// TIA Portal project "FESTO_SORTING_AND_DISTRIBUTING_STATION_WITH_HMI_AND_SCALANCE_V17_1" (V17)

(* hardware
DEVICE "S71500/ET200MP station_1"  S7-1500 station
   slot 0: "Rail_0"  Rack  6ES7 590-1***0-0AA0
   slot 1: "Sorting Station"  CPU 1512C-1 PN  6ES7 512-1CK01-0AB0  V2.5
      slot 3: "CPU display_1"  6ES7591-1AA00-0AA0
      slot 32768: "PROFINET interface_1"  X1
         slot 32769: "Port_1"  X1 P1
         slot 32770: "Port_2"  X1 P2
DEVICE "S71500/ET200MP station_2"  S7-1500 station
   slot 0: "Rail_0"  Rack  6ES7 590-1***0-0AA0
   slot 1: "Distributing Station"  CPU 1512C-1 PN  6ES7 512-1CK01-0AB0  V2.5
      slot 3: "CPU display_1"  6ES7591-1AA00-0AA0
      slot 32768: "PROFINET interface_1"  X1
         slot 32769: "Port_1"  X1 P1
         slot 32770: "Port_2"  X1 P2
DEVICE "HMI_1"  TP700 Comfort
   slot 0: "HMI_1"  TP700 Comfort  6AV2 124-0GC01-0AX0  16.0.0.0
   slot 1: "HMI_RT_1"  TP700 Comfort  6AV2 124-0GC01-0AX0  16.0.0.0
   slot 5: "HMI_1.IE_CP_1"  PROFINET Interface  16.0.0.0
      slot 1: "PROFINET Interface_1"  PROFINET Interface
         slot 1: "Port_1"  Port
         slot 2: "Port_2"  Port
   slot 7: "HMI_1.MPI/DP_CP_1"  MPI/DP Interface  16.0.0.0
*)

// ===== PLC "Sorting Station"  CPU 1512C-1 PN =====

VAR_GLOBAL   // PLC tag table "Default tag table"
   "ITEM_COUNTER_(PHOTOELECTRIC)" AT %I1.0 : Bool;
   "SORTER_EXTENDED_(INDUCTIVE)" AT %I1.1 : Bool;
   "CONVEYER" AT %Q5.2 : Bool;
   "SORTER" AT %Q5.0 : Bool;
   "START" AT %I0.0 : Bool;
   "STOP" AT %I0.1 : Bool;
   "AUTO" AT %I0.2 : Bool;
   "RESET" AT %I0.3 : Bool;
   "HMI_START" AT %M20.0 : Bool;
   "HMI_STOP" AT %M20.1 : Bool;
   "HMI_RESET" AT %M20.2 : Bool;
   "HMI_AUTO" AT %M20.3 : Bool;
   "POWER" AT %M0.0 : Bool;
   "BLACK_PART_MEM" AT %M40.0 : Bool;
   "PINK_PART_MEM" AT %M40.1 : Bool;
   "Clock_Byte" AT %MB300 : Byte;
   "Clock_10Hz" AT %M300.0 : Bool;
   "Clock_5Hz" AT %M300.1 : Bool;
   "Clock_2.5Hz" AT %M300.2 : Bool;
   "Clock_2Hz" AT %M300.3 : Bool;
   "Clock_1.25Hz" AT %M300.4 : Bool;
   "Clock_1Hz" AT %M300.5 : Bool;
   "Clock_0.625Hz" AT %M300.6 : Bool;
   "Clock_0.5Hz" AT %M300.7 : Bool;
   "Tag_1" AT %M40.2 : Bool;
   "RESTART_MEM" AT %M40.4 : Bool;
END_VAR

DATA_BLOCK "STEPS"   // DB2
{ S7_Optimized_Access := 'TRUE' }
VERSION : 0.1
   VAR
      Current_Step : Int;
   END_VAR
BEGIN
END_DATA_BLOCK

// folder: System blocks/Program resources

DATA_BLOCK "IEC_Timer_0_DB"   // DB3
{ S7_Optimized_Access := 'TRUE' }
AUTHOR : Simatic
FAMILY : IEC
NAME : IEC_TMR
VERSION : 1.0
// stored: InstanceOfName IEC_TIMER
"IEC_TIMER"
BEGIN
END_DATA_BLOCK

// folder: (top level)

ORGANIZATION_BLOCK "Sorting"   // OB1, LAD, ProgramCycle
TITLE = "Main Program Sweep (Cycle)"
{ S7_Optimized_Access := 'TRUE' }
VERSION : 0.1
   VAR_INPUT
      Initial_Call : Bool;   // Initial call of this OB
      Remanence : Bool;   // =True, if remanent data are available
   END_VAR
   VAR_TEMP   // added for the SCL form of the ladder/FBD networks
      _w1 : Bool;
      _w2 : Bool;
      _w3 : Bool;
   END_VAR
BEGIN

REGION Network 1
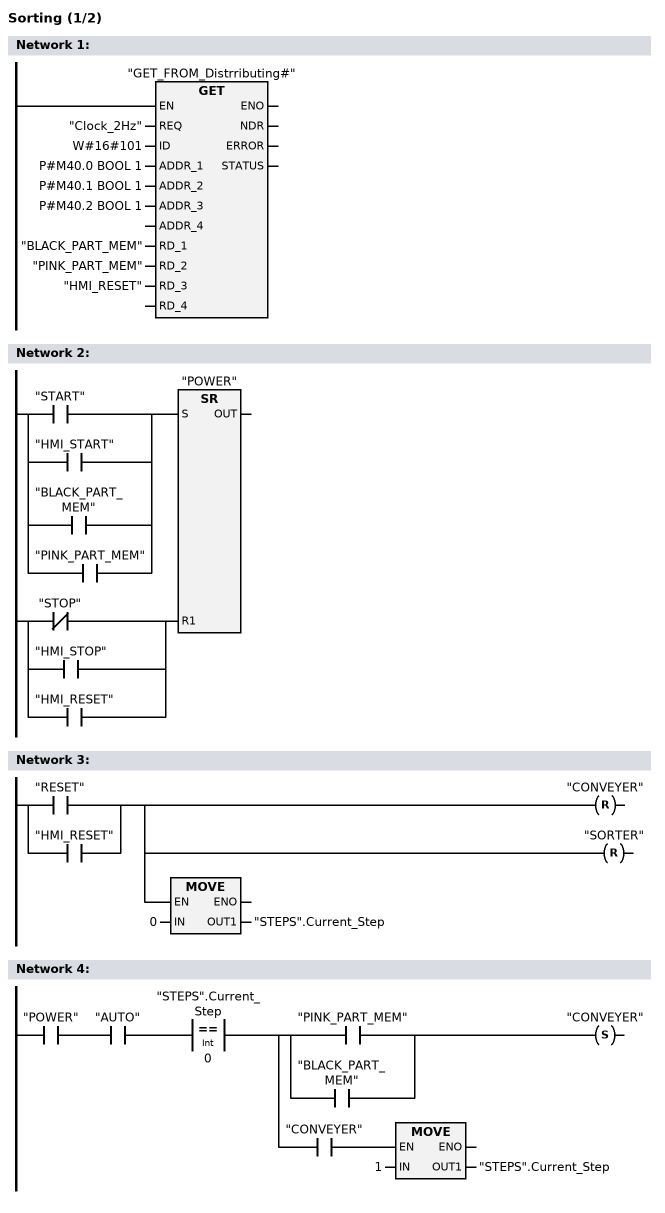
   "GET_FROM_Distrributing#"(REQ := "Clock_2Hz",   // GET
                           ID := W#16#101,
                           ADDR_1 := P#M40.0 BOOL 1,
                           ADDR_2 := P#M40.1 BOOL 1,
                           ADDR_3 := P#M40.2 BOOL 1,
                           RD_1 := "BLACK_PART_MEM",
                           RD_2 := "PINK_PART_MEM",
                           RD_3 := "HMI_RESET");
END_REGION

REGION Network 2
   RUNG wire#powerrail
      Contact( "START" )
      wire#w1
      S_SR(operand := "POWER", r1 := wire#w2)
   END_RUNG
   RUNG wire#powerrail
      Contact( "HMI_START" )
   END_RUNG wire#w1
   RUNG wire#powerrail
      Contact( "BLACK_PART_MEM" )
   END_RUNG wire#w1
   RUNG wire#powerrail
      Contact( "PINK_PART_MEM" )
   END_RUNG wire#w1
   RUNG wire#powerrail
      I_Contact( "STOP" )
   END_RUNG wire#w2
   RUNG wire#powerrail
      Contact( "HMI_STOP" )
   END_RUNG wire#w2
   RUNG wire#powerrail
      Contact( "HMI_RESET" )
   END_RUNG wire#w2
   // the same network as SCL:
   IF "START" OR "HMI_START" OR "BLACK_PART_MEM" OR "PINK_PART_MEM" THEN
       "POWER" := TRUE;   // SR flip-flop
   END_IF;
   IF NOT "STOP" OR "HMI_STOP" OR "HMI_RESET" THEN "POWER" := FALSE; END_IF;
END_REGION

REGION Network 3
   RUNG wire#powerrail
      Contact( "RESET" )
      wire#w1
      R_Coil( "CONVEYER" )
   END_RUNG
   RUNG wire#powerrail
      Contact( "HMI_RESET" )
   END_RUNG wire#w1
   RUNG wire#w1
      R_Coil( "SORTER" )
   END_RUNG
   RUNG wire#w1
      Move(in := 0, out1 => "STEPS".Current_Step)
   END_RUNG
   // the same network as SCL:
   IF "RESET" OR "HMI_RESET" THEN
       "CONVEYER" := FALSE;
       "SORTER" := FALSE;
       "STEPS".Current_Step := 0;
   END_IF;
END_REGION

REGION Network 4
   RUNG wire#powerrail
      Contact( "POWER" )
      Contact( "AUTO" )
      { S7_Templates := "SrcType := Int" } EQ_Contact(in1 := "STEPS".Current_Step, in2 := 0)
      wire#w1
      Contact( "PINK_PART_MEM" )
      wire#w2
      S_Coil( "CONVEYER" )
   END_RUNG
   RUNG wire#w1
      Contact( "BLACK_PART_MEM" )
   END_RUNG wire#w2
   RUNG wire#w1
      Contact( "CONVEYER" )
      Move(in := 1, out1 => "STEPS".Current_Step)
   END_RUNG
   // the same network as SCL:
   #_w1 := "POWER" AND "AUTO" AND ("STEPS".Current_Step = 0);
   IF #_w1 AND ("PINK_PART_MEM" OR "BLACK_PART_MEM") THEN "CONVEYER" := TRUE; END_IF;
   IF #_w1 AND "CONVEYER" THEN "STEPS".Current_Step := 1; END_IF;
END_REGION

REGION Network 5
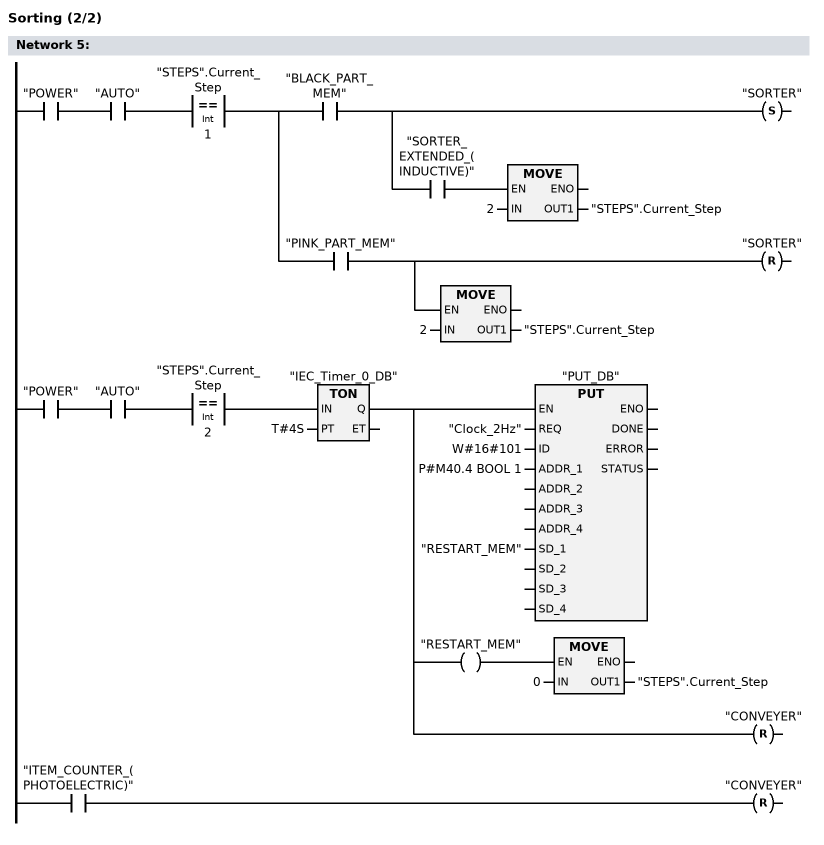
   #_w1 := "POWER" AND "AUTO" AND ("STEPS".Current_Step = 1);
   #_w2 := #_w1 AND "BLACK_PART_MEM";
   IF #_w2 THEN "SORTER" := TRUE; END_IF;
   IF #_w2 AND "SORTER_EXTENDED_(INDUCTIVE)" THEN "STEPS".Current_Step := 2; END_IF;
   IF #_w1 AND "PINK_PART_MEM" THEN
       "SORTER" := FALSE;
       "STEPS".Current_Step := 2;
   END_IF;
   "IEC_Timer_0_DB".TON(IN := "POWER" AND "AUTO" AND ("STEPS".Current_Step = 2), PT := T#4S);
   #_w3 := "IEC_Timer_0_DB".Q;
   IF #_w3 THEN
       "PUT_DB"(REQ := "Clock_2Hz", ID := W#16#101, ADDR_1 := P#M40.4 BOOL 1, SD_1 := "RESTART_MEM");   // PUT
   END_IF;
   "RESTART_MEM" := #_w3;
   IF #_w3 THEN
       "STEPS".Current_Step := 0;
       "CONVEYER" := FALSE;
   END_IF;
   IF "ITEM_COUNTER_(PHOTOELECTRIC)" THEN "CONVEYER" := FALSE; END_IF;
END_REGION
END_ORGANIZATION_BLOCK

// ===== PLC "Distributing Station"  CPU 1512C-1 PN =====

VAR_GLOBAL   // PLC tag table "Default tag table"
   "START" AT %I0.0 : Bool;
   "STOP" AT %I0.1 : Bool;
   "AUTO" AT %I0.2 : Bool;
   "RESET" AT %I0.3 : Bool;
   "PART_PRESENT(SORTING)" AT %I1.4 : Bool;
   "PHOTOELECTRIC(differentiate btwn black and pink)" AT %I1.7 : Bool;
   "INDUCTIVE(metallic and non-metallic" AT %I1.6 : Bool;
   "FEED_CYLINDER_EXTENDED" AT %I1.0 : Bool;
   "SORTER_EXTENDED" AT %I1.3 : Bool;
   "PART_PRESENT(FEED_CYLINDER)" AT %I1.2 : Bool;
   "HMI_START" AT %M0.0 : Bool;
   "HMI_STOP" AT %M0.1 : Bool;
   "HMI_AUTO" AT %M0.2 : Bool;
   "HMI_RESET" AT %M0.3 : Bool;
   "POWER" AT %M100.0 : Bool;
   "AUTO_MEM" AT %M100.1 : Bool;
   "CONVEYER_BACKWARD" AT %Q5.3 : Bool;
   "EXTEND_FEED_CYLINDER" AT %Q5.1 : Bool;
   "SORTER" AT %Q5.2 : Bool;
   "CONVEYER_FORWARD" AT %Q5.0 : Bool;
   "PART_HOLDER" AT %Q5.5 : Bool;
   "BLACK_MEM" AT %M40.0 : Bool;
   "PINK_MEM" AT %M40.1 : Bool;
   "Clock_Byte" AT %MB300 : Byte;
   "Clock_10Hz" AT %M300.0 : Bool;
   "Clock_5Hz" AT %M300.1 : Bool;
   "Clock_2.5Hz" AT %M300.2 : Bool;
   "Clock_2Hz" AT %M300.3 : Bool;
   "Clock_1.25Hz" AT %M300.4 : Bool;
   "Clock_1Hz" AT %M300.5 : Bool;
   "Clock_0.625Hz" AT %M300.6 : Bool;
   "Clock_0.5Hz" AT %M300.7 : Bool;
   "HMI_LED_RESET" AT %M100.4 : Bool;
   "STOP_MEM" AT %M100.5 : Bool;
   "RESET_MEM" AT %M40.2 : Bool;
   "Tag_1" AT %M20.2 : Bool;
   "RESTART_MEM" AT %M40.4 : Bool;
END_VAR

DATA_BLOCK "STEPS"   // DB1
{ S7_Optimized_Access := 'TRUE' }
VERSION : 0.1
   VAR
      Current_Steps : Real;
   END_VAR
BEGIN
END_DATA_BLOCK

// folder: System blocks/Program resources

DATA_BLOCK "#"   // DB2
{ S7_Optimized_Access := 'TRUE' }
AUTHOR : Simatic
FAMILY : IEC
NAME : IEC_TMR
VERSION : 1.0
// stored: InstanceOfName IEC_TIMER
"IEC_TIMER"
BEGIN
END_DATA_BLOCK

DATA_BLOCK "IEC_Timer_0_DB"   // DB5
{ S7_Optimized_Access := 'TRUE' }
AUTHOR : Simatic
FAMILY : IEC
NAME : IEC_TMR
VERSION : 1.0
// stored: InstanceOfName IEC_TIMER
"IEC_TIMER"
BEGIN
END_DATA_BLOCK

DATA_BLOCK "IEC_Timer_0_DB_1"   // DB8
{ S7_Optimized_Access := 'TRUE' }
AUTHOR : Simatic
FAMILY : IEC
NAME : IEC_TMR
VERSION : 1.0
// stored: InstanceOfName IEC_TIMER
"IEC_TIMER"
BEGIN
END_DATA_BLOCK

DATA_BLOCK "IEC_Timer_0_DB_2"   // DB9
{ S7_Optimized_Access := 'TRUE' }
AUTHOR : Simatic
FAMILY : IEC
NAME : IEC_TMR
VERSION : 1.0
// stored: InstanceOfName IEC_TIMER
"IEC_TIMER"
BEGIN
END_DATA_BLOCK

// folder: (top level)

ORGANIZATION_BLOCK "Distributing"   // OB1, LAD, ProgramCycle
TITLE = "Main Program Sweep (Cycle)"
{ S7_Optimized_Access := 'TRUE' }
VERSION : 0.1
   VAR_INPUT
      Initial_Call : Bool;   // Initial call of this OB
      Remanence : Bool;   // =True, if remanent data are available
   END_VAR
   VAR_TEMP   // added for the SCL form of the ladder/FBD networks
      _w1 : Bool;
      _w2 : Bool;
   END_VAR
BEGIN

REGION Network 1
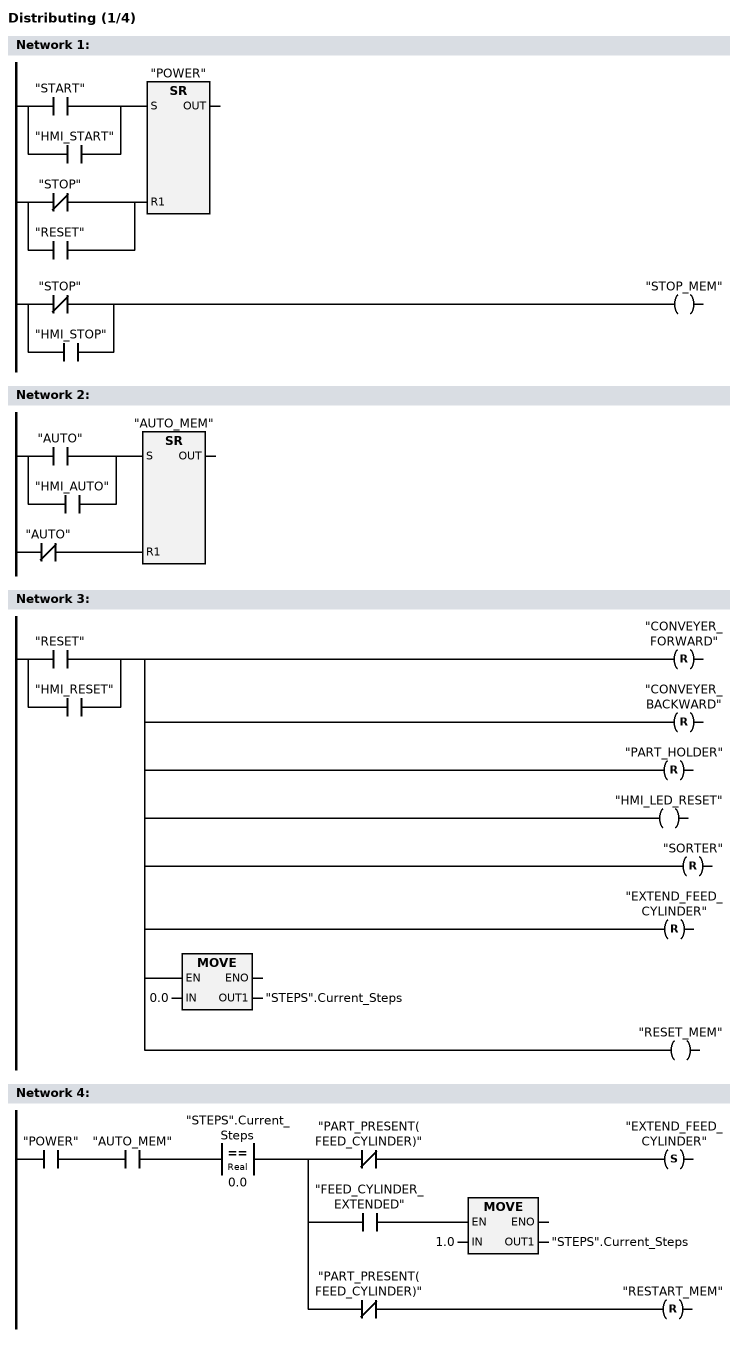
   RUNG wire#powerrail
      Contact( "START" )
      wire#w1
      S_SR(operand := "POWER", r1 := wire#w2)
   END_RUNG
   RUNG wire#powerrail
      Contact( "HMI_START" )
   END_RUNG wire#w1
   RUNG wire#powerrail
      I_Contact( "STOP" )
   END_RUNG wire#w2
   RUNG wire#powerrail
      Contact( "RESET" )
   END_RUNG wire#w2
   RUNG wire#powerrail
      I_Contact( "STOP" )
      wire#w3
      Coil( "STOP_MEM" )
   END_RUNG
   RUNG wire#powerrail
      Contact( "HMI_STOP" )
   END_RUNG wire#w3
   // the same network as SCL:
   IF "START" OR "HMI_START" THEN
       "POWER" := TRUE;   // SR flip-flop
   END_IF;
   IF NOT "STOP" OR "RESET" THEN "POWER" := FALSE; END_IF;
   "STOP_MEM" := NOT "STOP" OR "HMI_STOP";
END_REGION

REGION Network 2
   RUNG wire#powerrail
      Contact( "AUTO" )
      wire#w1
      S_SR(operand := "AUTO_MEM", r1 := wire#w2)
   END_RUNG
   RUNG wire#powerrail
      Contact( "HMI_AUTO" )
   END_RUNG wire#w1
   RUNG wire#powerrail
      I_Contact( "AUTO" )
   END_RUNG wire#w2
   // the same network as SCL:
   IF "AUTO" OR "HMI_AUTO" THEN
       "AUTO_MEM" := TRUE;   // SR flip-flop
   END_IF;
   IF NOT "AUTO" THEN "AUTO_MEM" := FALSE; END_IF;
END_REGION

REGION Network 3
   RUNG wire#powerrail
      Contact( "RESET" )
      wire#w1
      R_Coil( "CONVEYER_FORWARD" )
   END_RUNG
   RUNG wire#powerrail
      Contact( "HMI_RESET" )
   END_RUNG wire#w1
   RUNG wire#w1
      R_Coil( "CONVEYER_BACKWARD" )
   END_RUNG
   RUNG wire#w1
      R_Coil( "PART_HOLDER" )
   END_RUNG
   RUNG wire#w1
      Coil( "HMI_LED_RESET" )
   END_RUNG
   RUNG wire#w1
      R_Coil( "SORTER" )
   END_RUNG
   RUNG wire#w1
      R_Coil( "EXTEND_FEED_CYLINDER" )
   END_RUNG
   RUNG wire#w1
      Move(in := 0.0, out1 => "STEPS".Current_Steps)
   END_RUNG
   RUNG wire#w1
      Coil( "RESET_MEM" )
   END_RUNG
   // the same network as SCL:
   #_w1 := "RESET" OR "HMI_RESET";
   IF #_w1 THEN
       "CONVEYER_FORWARD" := FALSE;
       "CONVEYER_BACKWARD" := FALSE;
       "PART_HOLDER" := FALSE;
   END_IF;
   "HMI_LED_RESET" := #_w1;
   IF #_w1 THEN
       "SORTER" := FALSE;
       "EXTEND_FEED_CYLINDER" := FALSE;
       "STEPS".Current_Steps := 0.0;
   END_IF;
   "RESET_MEM" := #_w1;
END_REGION

REGION Network 4
   RUNG wire#powerrail
      Contact( "POWER" )
      Contact( "AUTO_MEM" )
      { S7_Templates := "SrcType := Real" } EQ_Contact(in1 := "STEPS".Current_Steps, in2 := 0.0)
      wire#w1
      I_Contact( "PART_PRESENT(FEED_CYLINDER)" )
      S_Coil( "EXTEND_FEED_CYLINDER" )
   END_RUNG
   RUNG wire#w1
      Contact( "FEED_CYLINDER_EXTENDED" )
      Move(in := 1.0, out1 => "STEPS".Current_Steps)
   END_RUNG
   RUNG wire#w1
      I_Contact( "PART_PRESENT(FEED_CYLINDER)" )
      R_Coil( "RESTART_MEM" )
   END_RUNG
   // the same network as SCL:
   #_w1 := "POWER" AND "AUTO_MEM" AND ("STEPS".Current_Steps = 0.0);
   IF #_w1 AND NOT "PART_PRESENT(FEED_CYLINDER)" THEN "EXTEND_FEED_CYLINDER" := TRUE; END_IF;
   IF #_w1 AND "FEED_CYLINDER_EXTENDED" THEN "STEPS".Current_Steps := 1.0; END_IF;
   IF #_w1 AND NOT "PART_PRESENT(FEED_CYLINDER)" THEN "RESTART_MEM" := FALSE; END_IF;
END_REGION

REGION Network 5
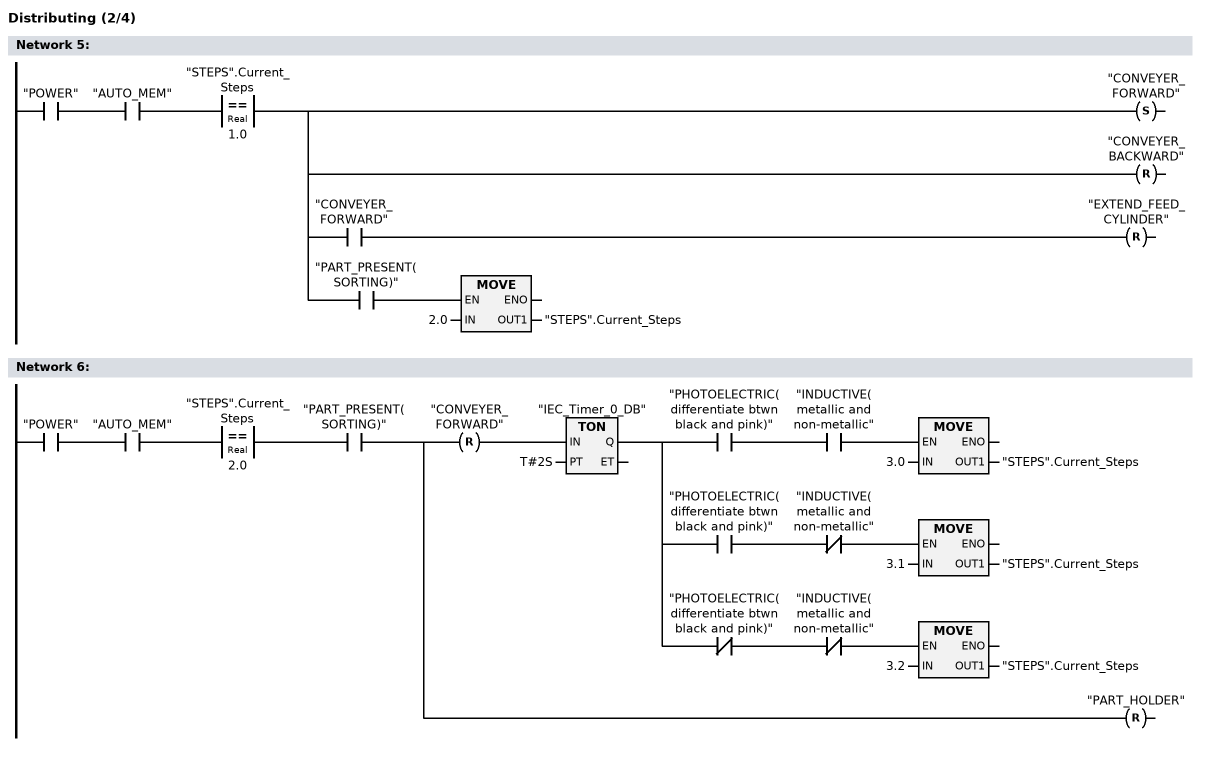
   RUNG wire#powerrail
      Contact( "POWER" )
      Contact( "AUTO_MEM" )
      { S7_Templates := "SrcType := Real" } EQ_Contact(in1 := "STEPS".Current_Steps, in2 := 1.0)
      wire#w1
      S_Coil( "CONVEYER_FORWARD" )
   END_RUNG
   RUNG wire#w1
      R_Coil( "CONVEYER_BACKWARD" )
   END_RUNG
   RUNG wire#w1
      Contact( "CONVEYER_FORWARD" )
      R_Coil( "EXTEND_FEED_CYLINDER" )
   END_RUNG
   RUNG wire#w1
      Contact( "PART_PRESENT(SORTING)" )
      Move(in := 2.0, out1 => "STEPS".Current_Steps)
   END_RUNG
   // the same network as SCL:
   #_w1 := "POWER" AND "AUTO_MEM" AND ("STEPS".Current_Steps = 1.0);
   IF #_w1 THEN
       "CONVEYER_FORWARD" := TRUE;
       "CONVEYER_BACKWARD" := FALSE;
   END_IF;
   IF #_w1 AND "CONVEYER_FORWARD" THEN "EXTEND_FEED_CYLINDER" := FALSE; END_IF;
   IF #_w1 AND "PART_PRESENT(SORTING)" THEN "STEPS".Current_Steps := 2.0; END_IF;
END_REGION

REGION Network 6
   #_w1 := "POWER" AND "AUTO_MEM" AND ("STEPS".Current_Steps = 2.0) AND "PART_PRESENT(SORTING)";
   IF #_w1 THEN "CONVEYER_FORWARD" := FALSE; END_IF;
   "IEC_Timer_0_DB".TON(IN := #_w1, PT := T#2S);
   IF "IEC_Timer_0_DB".Q AND "PHOTOELECTRIC(differentiate btwn black and pink)" AND "INDUCTIVE(metallic and non-metallic" THEN
       "STEPS".Current_Steps := 3.0;
   END_IF;
   IF "IEC_Timer_0_DB".Q AND "PHOTOELECTRIC(differentiate btwn black and pink)" AND NOT "INDUCTIVE(metallic and non-metallic" THEN
       "STEPS".Current_Steps := 3.1;
   END_IF;
   IF "IEC_Timer_0_DB".Q AND NOT "PHOTOELECTRIC(differentiate btwn black and pink)" AND NOT "INDUCTIVE(metallic and non-metallic" THEN
       "STEPS".Current_Steps := 3.2;
   END_IF;
   IF #_w1 THEN "PART_HOLDER" := FALSE; END_IF;
END_REGION

REGION Network 7
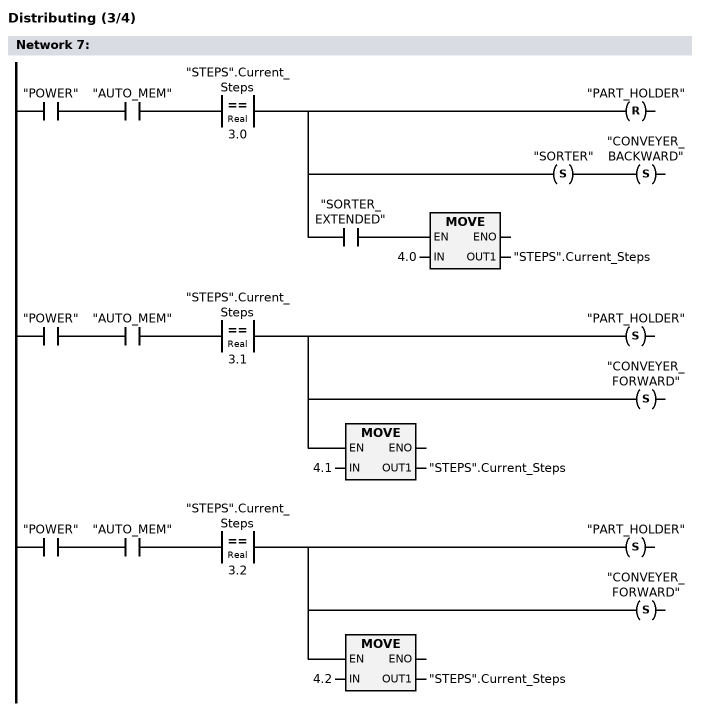
   RUNG wire#powerrail
      Contact( "POWER" )
      Contact( "AUTO_MEM" )
      { S7_Templates := "SrcType := Real" } EQ_Contact(in1 := "STEPS".Current_Steps, in2 := 3.0)
      wire#w1
      R_Coil( "PART_HOLDER" )
   END_RUNG
   RUNG wire#w1
      S_Coil( "SORTER" )
      S_Coil( "CONVEYER_BACKWARD" )
   END_RUNG
   RUNG wire#w1
      Contact( "SORTER_EXTENDED" )
      Move(in := 4.0, out1 => "STEPS".Current_Steps)
   END_RUNG
   RUNG wire#powerrail
      Contact( "POWER" )
      Contact( "AUTO_MEM" )
      { S7_Templates := "SrcType := Real" } EQ_Contact(in1 := "STEPS".Current_Steps, in2 := 3.1)
      wire#w2
      S_Coil( "PART_HOLDER" )
   END_RUNG
   RUNG wire#w2
      S_Coil( "CONVEYER_FORWARD" )
   END_RUNG
   RUNG wire#w2
      Move(in := 4.1, out1 => "STEPS".Current_Steps)
   END_RUNG
   RUNG wire#powerrail
      Contact( "POWER" )
      Contact( "AUTO_MEM" )
      { S7_Templates := "SrcType := Real" } EQ_Contact(in1 := "STEPS".Current_Steps, in2 := 3.2)
      wire#w3
      S_Coil( "PART_HOLDER" )
   END_RUNG
   RUNG wire#w3
      S_Coil( "CONVEYER_FORWARD" )
   END_RUNG
   RUNG wire#w3
      Move(in := 4.2, out1 => "STEPS".Current_Steps)
   END_RUNG
   // the same network as SCL:
   #_w1 := "POWER" AND "AUTO_MEM" AND ("STEPS".Current_Steps = 3.0);
   IF #_w1 THEN
       "PART_HOLDER" := FALSE;
       "SORTER" := TRUE;
       "CONVEYER_BACKWARD" := TRUE;
   END_IF;
   IF #_w1 AND "SORTER_EXTENDED" THEN "STEPS".Current_Steps := 4.0; END_IF;
   IF "POWER" AND "AUTO_MEM" AND ("STEPS".Current_Steps = 3.1) THEN
       "PART_HOLDER" := TRUE;
       "CONVEYER_FORWARD" := TRUE;
       "STEPS".Current_Steps := 4.1;
   END_IF;
   IF "POWER" AND "AUTO_MEM" AND ("STEPS".Current_Steps = 3.2) THEN
       "PART_HOLDER" := TRUE;
       "CONVEYER_FORWARD" := TRUE;
       "STEPS".Current_Steps := 4.2;
   END_IF;
END_REGION

REGION Network 8
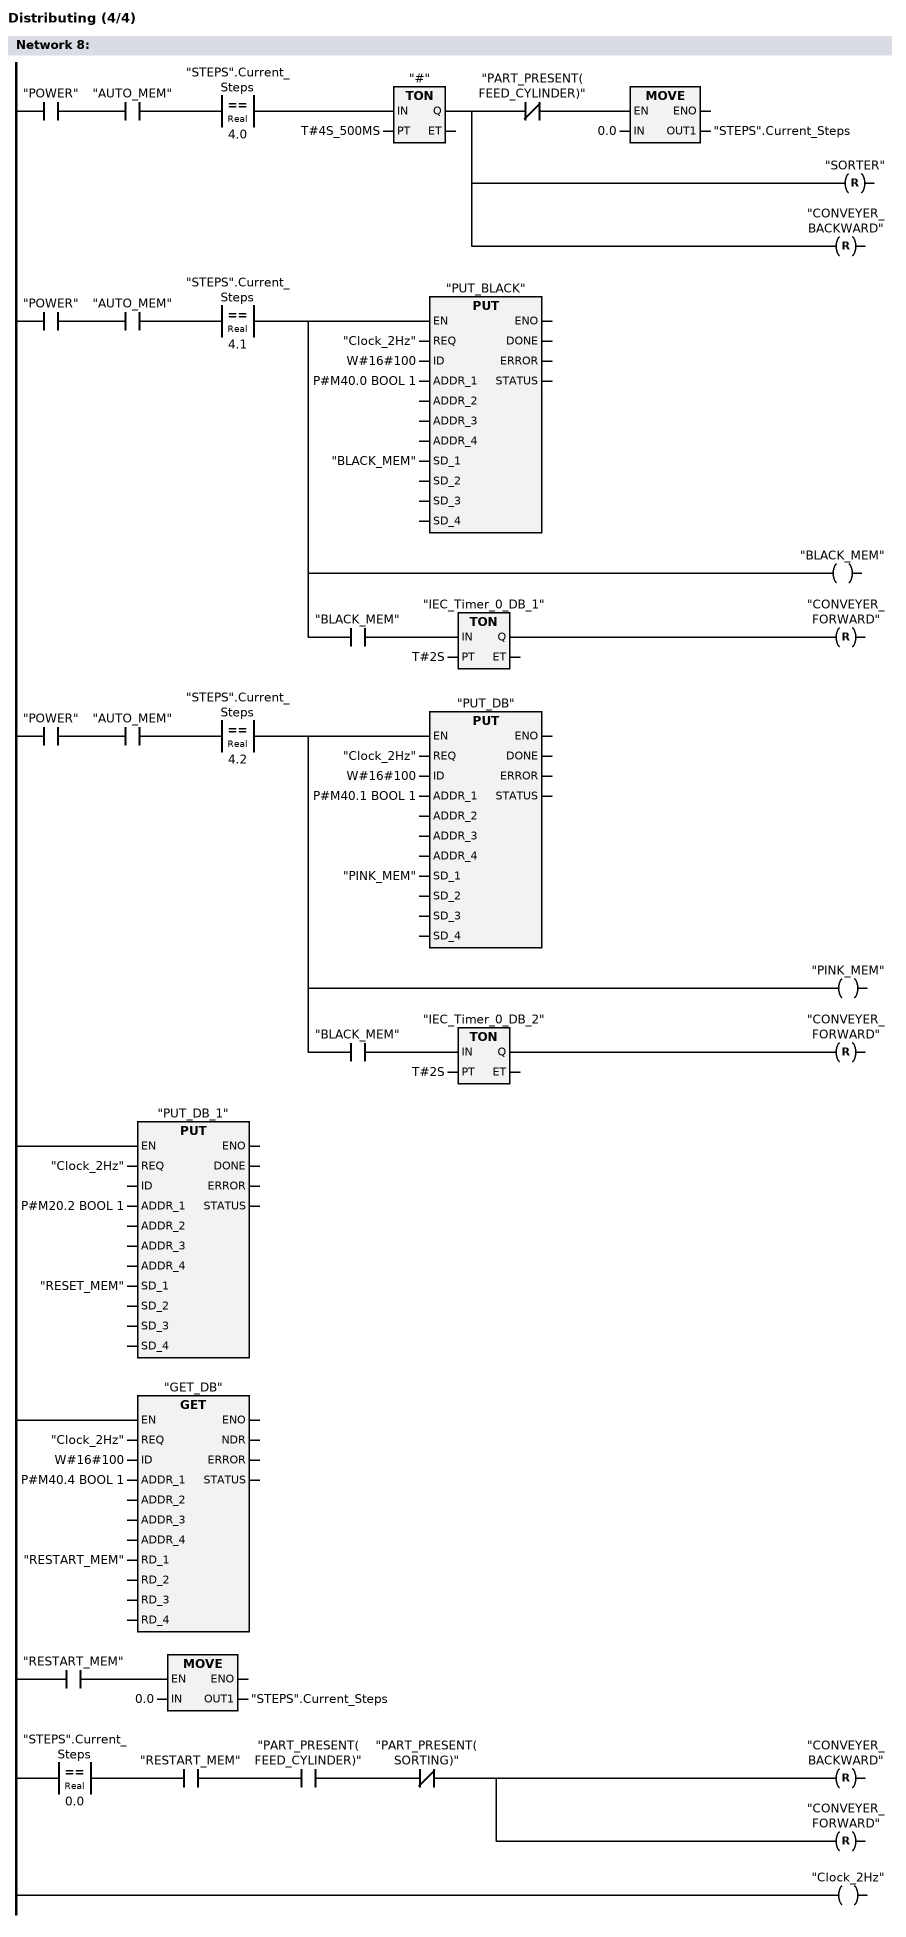
   "#".TON(IN := "POWER" AND "AUTO_MEM" AND ("STEPS".Current_Steps = 4.0), PT := T#4S_500MS);
   IF "#".Q AND NOT "PART_PRESENT(FEED_CYLINDER)" THEN "STEPS".Current_Steps := 0.0; END_IF;
   IF "#".Q THEN
       "SORTER" := FALSE;
       "CONVEYER_BACKWARD" := FALSE;
   END_IF;
   #_w1 := "POWER" AND "AUTO_MEM" AND ("STEPS".Current_Steps = 4.1);
   IF #_w1 THEN
       "PUT_BLACK"(REQ := "Clock_2Hz", ID := W#16#100, ADDR_1 := P#M40.0 BOOL 1, SD_1 := "BLACK_MEM");   // PUT
   END_IF;
   "BLACK_MEM" := #_w1;
   "IEC_Timer_0_DB_1".TON(IN := #_w1 AND "BLACK_MEM", PT := T#2S);
   IF "IEC_Timer_0_DB_1".Q THEN "CONVEYER_FORWARD" := FALSE; END_IF;
   #_w2 := "POWER" AND "AUTO_MEM" AND ("STEPS".Current_Steps = 4.2);
   IF #_w2 THEN
       "PUT_DB"(REQ := "Clock_2Hz", ID := W#16#100, ADDR_1 := P#M40.1 BOOL 1, SD_1 := "PINK_MEM");   // PUT
   END_IF;
   "PINK_MEM" := #_w2;
   "IEC_Timer_0_DB_2".TON(IN := #_w2 AND "BLACK_MEM", PT := T#2S);
   IF "IEC_Timer_0_DB_2".Q THEN "CONVEYER_FORWARD" := FALSE; END_IF;
   "PUT_DB_1"(REQ := "Clock_2Hz", ADDR_1 := P#M20.2 BOOL 1, SD_1 := "RESET_MEM");   // PUT
   "GET_DB"(REQ := "Clock_2Hz", ID := W#16#100, ADDR_1 := P#M40.4 BOOL 1, RD_1 := "RESTART_MEM");   // GET
   IF "RESTART_MEM" THEN "STEPS".Current_Steps := 0.0; END_IF;
   IF ("STEPS".Current_Steps = 0.0) AND "RESTART_MEM" AND "PART_PRESENT(FEED_CYLINDER)" AND NOT "PART_PRESENT(SORTING)" THEN
       "CONVEYER_BACKWARD" := FALSE;
       "CONVEYER_FORWARD" := FALSE;
   END_IF;
   "Clock_2Hz" := TRUE;
END_REGION
END_ORGANIZATION_BLOCK

(* ===== HMI "HMI_RT_1" =====
system functions are stored by id; their names below are inferred from use
connection "HMI_Connection_1": ETHERNET, S7_1500_OMS

HMI tags "Default tag table"
   "HMI_START" : Bool = PLC HMI_START AT %M0.0, 1 s
   "HMI_STOP" : Bool = PLC HMI_STOP AT %M0.1, 1 s
   "HMI_RESET" : Bool = PLC HMI_RESET AT %M0.3, 1 s
   "HMI_AUTO" : Bool = PLC HMI_AUTO AT %M0.2, 1 s
   "POWER" : Bool = PLC POWER AT %M100.0, 1 s
   "HMI_LED_RESET" : Bool = PLC HMI_LED_RESET AT %M100.4, 1 s
   "STOP_MEM" : Bool = PLC STOP_MEM AT %M100.5, 1 s

screen "Screen_1" 800x480
   Button "Button_1" at 29,115 size 95x57; TextOff 'Start'
      on Press: SetBit("HMI_START")
      on Release: ResetBit("HMI_START")
   Button "Button_2" at 158,115 size 95x57; TextOff 'Stop'
      on Press: SetBit("HMI_STOP")
      on Release: ResetBit("HMI_STOP")
   Button "Button_3" at 29,247 size 95x57; TextOff 'Reset'
      on Press: SetBit("HMI_RESET")
      on Release: ResetBit("HMI_RESET")
   Switch "Switch_1" at 168,245 size 238x59; CaptionText 'Switch'; TextOff 'OFF'; TextOn 'ON'
      on SwitchOn: SetBit("HMI_AUTO")
      on SwitchOff: ResetBit("HMI_AUTO")
   Circle "Circle_1" at 496,115 size 72x72
      Appearance <- "POWER"
   Circle "Circle_2" at 496,203 size 72x72
      Appearance <- "HMI_LED_RESET"
   Circle "Circle_3" at 496,291 size 72x72
      Appearance <- "STOP_MEM"
   TextField "Text field_1" at 611,129 size 40x25; Text 'Start'
   TextField "Text field_2" at 611,222 size 47x25; Text 'Reset'
   TextField "Text field_3" at 611,303 size 37x25; Text 'Stop'
*)